TYPE EventTestsystem :
STRUCT
  runner: EventRunner;
  event: FBEvent(runner);
END_STRUCT
END_TYPE

(* stored: Version 1.1.0.1, ProductVersion 3.1.4022.18
   DUT EventTestsystem: Id {1d1d3ef4-d20e-433d-90eb-bc663d6abd18} *)
